(* IEC 61131-3 sources: vscode-twincat-st/src/sample/Features, 1 file *)

(* ---- DocumentHighlightProvider.st ---- *)
// Goal: Highlight only semantically related tokens
FUNCTION_BLOCK FB_Highlight

    VAR
        highlight: INT;
    END_VAR

    METHOD M_Highlight

        VAR
            highlight: INT;
        END_VAR

        highlight := 1;
    END_METHOD
END_FUNCTION_BLOCK
